FUNCTION_BLOCK PAMTank EXTENDS PAProcessModule IMPLEMENTS IPAMSilo
VAR_INPUT
END_VAR
VAR_OUTPUT
END_VAR
VAR
	_PAPointMatIn1 : PAPoint(THIS^);
	_PAPointMatOut1 : PAPoint(THIS^);
END_VAR

METHOD FB_init : BOOL
VAR_INPUT
	bInitRetains : BOOL; // if TRUE, the retain variables are initialized (warm start / cold start)
	bInCopyCode : BOOL;  // if TRUE, the instance afterwards gets moved into the copy code (online change)
	parent : IACComponent;
END_VAR
AddPoint(_PAPointMatIn1);
AddPoint(_PAPointMatOut1);
END_METHOD

PROPERTY PUBLIC PAPointMatIn1 : IACPoint
GET
PAPointMatIn1 := _PAPointMatIn1;
END_GET
END_PROPERTY

PROPERTY PUBLIC PAPointMatOut1 : IACPoint
GET
PAPointMatOut1 := _PAPointMatOut1;
END_GET
END_PROPERTY

END_FUNCTION_BLOCK

(* stored: Version 1.1.0.1, ProductVersion 3.1.4020.12
   POU PAMTank: Id {4a663811-0f34-40a4-9bb8-615f716776a8}, SpecialFunc None
   Method FB_init: Id {6f5ff4eb-fa9e-4dba-8c14-b49c87e9e201}
   Property PAPointMatIn1: Id {51d95bba-e005-4438-874e-26ac7bc4e6fd}
   Get Get: Id {b1721566-9f56-4278-a448-9feb2acc9c34}
   Property PAPointMatOut1: Id {5b74935c-8520-48c4-babd-97f05252a8cf}
   Get Get: Id {c2d1f3c6-ca3c-42c8-8f51-005d594c14a0} *)
